(* IEC 61131-3 sources: gridguard_dtt/plc_logic/programs, 10 files *)

(* ---- breaker_auto_cycle.st ---- *)
(*
OpenPLC Automatic Breaker Cycling Program
Automatically cycles the breaker: CLOSED for 30s, OPEN for 10s
Perfect for testing anomaly detection systems
*)

PROGRAM breaker_auto_cycle
VAR
    circuit_breaker AT %QX0.0 : BOOL;
    cycle_counter AT %MD0 : DINT;
    cycle_limit AT %MD4 : DINT;
    closed_limit AT %MD8 : DINT;
END_VAR

(* Initialize constants on first run *)
IF cycle_limit = 0 THEN
    cycle_limit := 2000;
    closed_limit := 1500;
END_IF;

(* Increment counter *)
cycle_counter := cycle_counter + 1;

(* Reset counter when cycle completes *)
IF cycle_counter >= cycle_limit THEN
    cycle_counter := 0;
END_IF;

(* Breaker logic: CLOSED for first 30s, OPEN for last 10s *)
IF cycle_counter < closed_limit THEN
    circuit_breaker := TRUE;
ELSE
    circuit_breaker := FALSE;
END_IF;

END_PROGRAM

CONFIGURATION Config0
    RESOURCE Res0 ON PLC
        TASK task0(INTERVAL := T#20ms, PRIORITY := 0);
        PROGRAM instance0 WITH task0 : breaker_auto_cycle;
    END_RESOURCE
END_CONFIGURATION

(* ---- breaker_auto_cycle_simple.st ---- *)
(*
OpenPLC Automatic Breaker Cycling Program
Uses only simple boolean logic like breaker_control_complete.st
Cycles breaker: CLOSED most of the time, OPEN occasionally
*)

PROGRAM breaker_auto_cycle
VAR
    circuit_breaker AT %QX0.0 : BOOL;
    always_on AT %IX0.0 : BOOL;
END_VAR

(* Simple cycling logic: breaker follows input state *)
(* This will be controlled by SCADA simulation instead *)
circuit_breaker := always_on;

END_PROGRAM

CONFIGURATION Config0
    RESOURCE Res0 ON PLC
        TASK task0(INTERVAL := T#20ms, PRIORITY := 0);
        PROGRAM instance0 WITH task0 : breaker_auto_cycle;
    END_RESOURCE
END_CONFIGURATION

(* ---- breaker_bool_cycle.st ---- *)
(*
OpenPLC Automatic Breaker Cycling Program
Uses only BOOL variables to avoid INT declaration issues
Cycles breaker automatically without external inputs
*)

PROGRAM breaker_auto_cycle
VAR
    circuit_breaker AT %QX0.0 : BOOL;
    timer1 : BOOL;
    timer2 : BOOL;
    timer3 : BOOL;
    timer4 : BOOL;
    timer5 : BOOL;
END_VAR

(* Simple state machine using boolean cascade *)
(* This creates a slow cycling pattern *)
timer1 := NOT timer1;

IF timer1 THEN
    timer2 := NOT timer2;
END_IF;

IF timer2 THEN
    timer3 := NOT timer3;
END_IF;

IF timer3 THEN
    timer4 := NOT timer4;
END_IF;

IF timer4 THEN
    timer5 := NOT timer5;
END_IF;

(* Breaker follows timer5 with some logic for cycling *)
circuit_breaker := timer5 OR timer4;

END_PROGRAM

CONFIGURATION Config0
    RESOURCE Res0 ON PLC
        TASK task0(INTERVAL := T#20ms, PRIORITY := 0);
        PROGRAM instance0 WITH task0 : breaker_auto_cycle;
    END_RESOURCE
END_CONFIGURATION

(* ---- breaker_control.st ---- *)
PROGRAM breaker_control
VAR
    start_button AT %IX0.0 : BOOL;  (* Input - Start button *)
    circuit_breaker AT %QX0.0 : BOOL;  (* Output - Circuit breaker coil *)
END_VAR

(* Simple breaker control logic *)
(* When start button is pressed, energize circuit breaker *)
circuit_breaker := start_button;

END_PROGRAM

(* ---- breaker_control_complete.st ---- *)
(*
OpenPLC Breaker Control Program
This program implements simple breaker control logic equivalent to:
   | start_button |        ( circuit_breaker )
---|----] [-------|--------(---------------)---
   %IX0.0          %QX0.0
*)

PROGRAM breaker_control
VAR
    start_button AT %IX0.0 : BOOL;  (* Digital input - Start button *)
    circuit_breaker AT %QX0.0 : BOOL;  (* Digital output - Circuit breaker coil *)
END_VAR

(* Main control logic *)
(* Direct assignment: when start button is active, circuit breaker is energized *)
circuit_breaker := start_button;

END_PROGRAM

CONFIGURATION Config0
    RESOURCE Res0 ON PLC
        TASK task0(INTERVAL := T#20ms, PRIORITY := 0);
        PROGRAM instance0 WITH task0 : breaker_control;
    END_RESOURCE
END_CONFIGURATION

(* ---- breaker_control_interactive.st ---- *)
(*
OpenPLC Interactive Breaker Control Program
This program allows remote control of the circuit breaker via Modbus
- QX0.0: Circuit breaker output (controlled by logic)
- QX0.1: Manual control register (writable via Modbus)
- QX0.2: System status indicator
*)

PROGRAM breaker_control_interactive
VAR
    (* Inputs *)
    start_button AT %IX0.0 : BOOL;         (* Physical start button input *)

    (* Outputs *)
    circuit_breaker AT %QX0.0 : BOOL;      (* Circuit breaker coil *)
    manual_control AT %QX0.1 : BOOL;       (* Manual control flag (writable) *)
    system_active AT %QX0.2 : BOOL;        (* System status indicator *)

    (* Internal variables *)
    prev_manual_control : BOOL;            (* Previous state for edge detection *)
    breaker_state : BOOL;                  (* Internal breaker state *)
    manual_mode : BOOL;                    (* Manual mode flag *)
    toggle_trigger : BOOL;                 (* Toggle edge detection *)
END_VAR

(* Initialize on first scan *)
IF NOT system_active THEN
    system_active := TRUE;
    breaker_state := FALSE;
    manual_mode := FALSE;
    prev_manual_control := manual_control;
END_IF;

(* Detect rising edge on manual control for toggle operation *)
toggle_trigger := manual_control AND NOT prev_manual_control;
prev_manual_control := manual_control;

(* Toggle breaker state on manual control edge *)
IF toggle_trigger THEN
    breaker_state := NOT breaker_state;
    manual_mode := TRUE;
END_IF;

(* Auto mode: breaker follows start button *)
IF NOT manual_mode AND start_button THEN
    breaker_state := TRUE;
END_IF;

(* Output the breaker state *)
circuit_breaker := breaker_state;

(* Reset manual mode if start button is pressed *)
IF start_button THEN
    manual_mode := FALSE;
END_IF;

END_PROGRAM

CONFIGURATION Config0
    RESOURCE Res0 ON PLC
        TASK task0(INTERVAL := T#20ms, PRIORITY := 0);
        PROGRAM instance0 WITH task0 : breaker_control_interactive;
    END_RESOURCE
END_CONFIGURATION

(* ---- breaker_control_manual.st ---- *)
(*
OpenPLC Breaker Control with Manual Override
- IX0.0: Start button (auto mode)
- IX0.1: Manual mode enable
- QX0.0: Circuit breaker output
- QX0.1: Status indicator

Manual control via Modbus:
- Write to address 10001 (mapped to IX0.1) to enable manual mode
- When in manual mode, QX0.0 can be controlled via Modbus
*)

PROGRAM breaker_control_manual
VAR
    (* Inputs *)
    start_button AT %IX0.0 : BOOL;         (* Auto mode start button *)
    manual_enable AT %IX0.1 : BOOL;        (* Manual mode enable *)

    (* Outputs *)
    circuit_breaker AT %QX0.0 : BOOL;      (* Circuit breaker control *)
    status_led AT %QX0.1 : BOOL;           (* Status indicator *)

    (* Internal variables *)
    manual_mode : BOOL := FALSE;
    breaker_command : BOOL := FALSE;
    prev_manual_enable : BOOL := FALSE;
    manual_toggle : BOOL := FALSE;
END_VAR

(* Detect rising edge on manual enable for mode switching *)
manual_toggle := manual_enable AND NOT prev_manual_enable;
prev_manual_enable := manual_enable;

(* Switch to manual mode on rising edge *)
IF manual_toggle THEN
    manual_mode := NOT manual_mode;
END_IF;

(* Control logic *)
IF manual_mode THEN
    (* Manual mode: preserve current output state unless overridden *)
    (* The output can be controlled directly via Modbus writes to QX0.0 *)
    (* We don't override it here, letting manual control work *)
    status_led := TRUE;  (* Indicate manual mode *)
ELSE
    (* Auto mode: output follows start button *)
    circuit_breaker := start_button;
    status_led := start_button;  (* Status follows breaker in auto mode *)
END_IF;

END_PROGRAM

CONFIGURATION Config0
    RESOURCE Res0 ON PLC
        TASK task0(INTERVAL := T#100ms, PRIORITY := 0);
        PROGRAM instance0 WITH task0 : breaker_control_manual;
    END_RESOURCE
END_CONFIGURATION

(* ---- breaker_control_redteam_ready.st ---- *)
(*
GridGuard SCADA Red Team Testing PLC Program

Attack Vectors:
1. Emergency Bypass: Set bypass_active (QX0.5) = TRUE
2. Maintenance Mode: Write -559038737 to maint_key (MD12)
3. Timer Manipulation: Modify timer_preset (MD8)
*)

PROGRAM breaker_control_redteam_ready
VAR
    (* Located variables - I/O mapping *)
    start_btn AT %IX0.0 : BOOL;
    stop_btn AT %IX0.1 : BOOL;
    health_ok AT %IX0.2 : BOOL;
    breaker_out AT %QX0.0 : BOOL;
    status_led AT %QX0.1 : BOOL;
    fault_led AT %QX0.2 : BOOL;
    maint_led AT %QX0.3 : BOOL;
    alert_led AT %QX0.4 : BOOL;
    bypass_active AT %QX0.5 : BOOL;
    debug_active AT %QX0.6 : BOOL;
    counter AT %MD0 : DINT;
    event_count AT %MD4 : DINT;
    timer_preset AT %MD8 : DINT;
    maint_key AT %MD12 : DINT;

    (* Additional located variables *)
    breaker_state AT %QX0.7 : BOOL;
    safety_timer AT %MD16 : DINT;
    maint_mode AT %QX1.0 : BOOL;
END_VAR

    (* The program logic must begin AFTER the END_VAR block. *)

    (* Initialize on first run *)
    IF counter = 0 THEN
        timer_preset := 100;
        event_count := 0;
        maint_mode := FALSE;
        safety_timer := 0;
        breaker_state := TRUE;  (* Start with breaker CLOSED for red team testing *)
    END_IF;

    (* Increment counter *)
    counter := counter + 1;

    (* ATTACK VECTOR 1: Emergency Bypass *)
    IF bypass_active THEN
        breaker_state := start_btn;
        event_count := event_count + 1;
    ELSE
        (* Normal Operation - maintain closed state unless explicitly stopped *)
        IF start_btn THEN  (* Removed health_ok requirement *)
            IF safety_timer = 0 THEN
                safety_timer := timer_preset;
            END_IF;
        END_IF;

        IF safety_timer > 0 THEN
            safety_timer := safety_timer - 1;
            IF safety_timer = 0 AND start_btn THEN
                breaker_state := TRUE;
            END_IF;
        END_IF;

        (* Only open breaker if explicitly stopped or health explicitly fails *)
        IF stop_btn THEN
            breaker_state := FALSE;
            safety_timer := 0;
        (* Remove health_ok check since it defaults to FALSE when not connected *)
        (* ELSIF NOT health_ok THEN
            breaker_state := FALSE;
            safety_timer := 0; *)
        END_IF;
    END_IF;

    (* ATTACK VECTOR 2: Maintenance Override *)
    IF maint_key = -559038737 THEN
        maint_mode := TRUE;
        breaker_state := start_btn;
        event_count := event_count + 1;
    END_IF;

    (* Outputs *)
    breaker_out := breaker_state;
    status_led := breaker_state;
    fault_led := FALSE;  (* No health monitoring for now *)
    maint_led := maint_mode;
    alert_led := (event_count > 10);

END_PROGRAM

CONFIGURATION Config0
    RESOURCE Res0 ON PLC
        TASK task0(INTERVAL := T#20ms, PRIORITY := 0);
        PROGRAM instance0 WITH task0 : breaker_control_redteam_ready;
    END_RESOURCE
END_CONFIGURATION

(* ---- breaker_toggle_simple.st ---- *)
(*
OpenPLC Simple Toggle Breaker Control
Uses QX0.0 as both output and toggle input
- Write to QX0.0 to toggle the breaker state
*)

PROGRAM breaker_toggle
VAR
    circuit_breaker AT %QX0.0 : BOOL;      (* Circuit breaker - both input and output *)

    (* Internal variables for edge detection *)
    prev_state : BOOL := FALSE;
    internal_breaker : BOOL := FALSE;
    toggle_command : BOOL;
END_VAR

(* Read the current command from Modbus *)
toggle_command := circuit_breaker;

(* Detect rising edge (0->1 transition) for toggle *)
IF toggle_command AND NOT prev_state THEN
    internal_breaker := NOT internal_breaker;
END_IF;

(* Update previous state for next scan *)
prev_state := toggle_command;

(* Output the internal breaker state *)
circuit_breaker := internal_breaker;

END_PROGRAM

CONFIGURATION Config0
    RESOURCE Res0 ON PLC
        TASK task0(INTERVAL := T#50ms, PRIORITY := 0);
        PROGRAM instance0 WITH task0 : breaker_toggle;
    END_RESOURCE
END_CONFIGURATION

(* ---- main.st ---- *)
CONFIGURATION config
    RESOURCE resource1 ON PLC
        TASK main_task(INTERVAL := T#100ms, PRIORITY := 0);
        PROGRAM instance0 WITH main_task : breaker_control;
    END_RESOURCE
END_CONFIGURATION
